FUNCTION F_RemoveSign : STRING(255)
(**************************************************************************************
 * 	Application		:	BoxControl Framework
 *	Revision		:	$Revision: 404529 $
 *	Revision date	:	$Date: 2018-04-23 08:21:38 +0200 (Mo., 23 Apr 2018) $
 *	Last changed by	:	$Author: b7bolm $
 *	URL				:	$URL: http://almscdc.swisslog.com/repo/SWPD/Development/BoxControlFramework/20_Release/trunk/01_Software/BCF/BCF/JumpStart/30_Toolbox/12_StringStream/F_RemoveSign.TcPOU $
 *
 *	Purpose			:	Remove a sign from a string.
 *
 * ------------------------------------------------------------------------------------
 *	Copyright Swisslog [IP AG], Switzerland. All rights reserved.
 * 
 * ------------------------------------------------------------------------------------
 *	
 * 	Revision History: 
 *
 * 	VERSION			DATE			INITIALS			DESCRIPTION
 *	0.1				01.01.2001		swl					Example
 *
 **************************************************************************************)
VAR_INPUT
	InputString		: STRING(255); // Input string
	Sign			: STRING(1); // Sign to remove
END_VAR
VAR
	Idx				: INT; // Iterator
	pASCII_Array	: POINTER TO ARRAY[1..255] OF BYTE;
	pSign			: POINTER TO BYTE;
	ASCII_Value		: INT; // Value
END_VAR

// Initialize
F_RemoveSign := '';

// Build ASCII array and sign as byte
pASCII_Array := ADR(InputString);
pSign := ADR(Sign);

// Go Through string
FOR Idx := 1 TO LEN(InputString) DO
	// Get first ASCII sign as INT
	ASCII_Value := BYTE_TO_INT(pASCII_Array^[Idx]);
	
	// Add all except sign to new string
	IF pSign^ <> ASCII_Value THEN
		// Build string
		fbFormatString( sFormat := '%C',
						arg1 	:= F_BYTE(pASCII_Array^[Idx]));
		
		// Return alpha numeric string
		F_RemoveSign := CONCAT(F_RemoveSign, fbFormatString.sOut);
	END_IF
END_FOR

END_FUNCTION

(* stored: Version 1.1.0.1, ProductVersion 3.1.4020.6
   POU F_RemoveSign: Id {7525b74e-8e17-4835-974f-38ae53f7f2fa}, SpecialFunc None *)
